// TIA Portal V18 export
// export: Created 2026-03-12T15:56:19.3301424Z, ExportSetting WithDefaults, DisplayName Totally Integrated Automation Portal, DisplayVersion V18 Update 5, DisplayName TIA Portal Openness, DisplayVersion V18 Update 5, DisplayName TIA Portal Version Control Interface, DisplayVersion V18, DisplayName SINAMICS Startdrive Advanced, DisplayVersion V18, DisplayName SINAMICS Startdrive G130, G150, S120, S150, SINAMICS MV, S210, DisplayVersion V18, DisplayName SINAMICS Startdrive G110M, G120, G120C, G120D, G120P, G115D, DisplayVersion V18, DisplayName STEP 7 Professional, DisplayVersion V18 Update 5, DisplayName STEP 7 Safety, DisplayVersion V18, DisplayName WinCC Professional, DisplayVersion V18 Update 5
DATA_BLOCK "FB PROCESSO_AUTO_ELEVATORIA_BH-01"   // DB772
VERSION : 0.1
// stored: AutoNumber true, DBAccessibleFromOPCUA true, DBAccessibleFromWebserver true, InstanceOfName FB PROCESSO_AUTO_ELEVATORIA, InstanceOfType FB
"FB PROCESSO_AUTO_ELEVATORIA"
   // VAR_INPUT
   //    INPUT_HABILITA_PAR : Bool;
   //    INPUT_REMOTO_AUTO_A : Bool;
   //    INPUT_REMOTO_AUTO_B : Bool;
   //    INPUT_COMANDO_ALTERNANCIA_ATIVO : Bool;
   //    INPUT_FALHA_BOMBA_A : Bool;
   //    INPUT_FALHA_BOMBA_B : Bool;
   //    INPUT_CADASTRO_TEMPO_LIGADO_A : Real;
   //    INPUT_CADASTRO_TEMPO_LIGADO_B : Real;
   //    INPUT_STATUS_SENSOR : Real;
   //    INPUT_CADASTRO_LIGA_A : Real;
   //    INPUT_CADASTRO_DESLIGA_A : Real;
   //    INPUT_CADASTRO_LIGA_B : Real;
   //    INPUT_CADASTRO_DESLIGA_B : Real;
   // END_VAR
   // VAR_OUTPUT
   //    HORA_ALTERNANCIA_A : Real;
   //    HORA_ALTERNANCIA_B : Real;
   //    HABILITA_LIGA_BOMBA_A : Bool;
   //    HABILITA_LIGA_BOMBA_B : Bool;
   // END_VAR
   // VAR
   //    "FB CONTADOR_A" { S7_SetPoint := 'True'} : "FB CONTADOR";
   //    "FB CONTADOR_B" { S7_SetPoint := 'True'} : "FB CONTADOR";
   // END_VAR
BEGIN
END_DATA_BLOCK
